(* PLC project FBD_EVOLUTION_1, Beckhoff Automation GmbH TwinCAT PLC Control 3.5.10.30 *)
(* stored: creationDateTime 2019-09-26T17:00:57.7902241, modificationDateTime 2019-09-26T17:00:57.7902241 *)

PROGRAM POU
VAR
	A: BOOL;
	B: BOOL;
	C: BOOL;
END_VAR

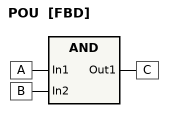
(* FBD diagram, written out as Structured Text *)
C := A AND B;
END_PROGRAM

CONFIGURATION Application
  RESOURCE FBD_EVOLUTION_1 ON PLC
(* global variable list GVL *)
{attribute 'qualified_only'}
VAR_GLOBAL
	IsSFCResetting : BOOL;
END_VAR
    TASK PlcTask(INTERVAL := T#0ms, PRIORITY := 20);
    PROGRAM Main WITH PlcTask : Main;
  END_RESOURCE
END_CONFIGURATION
